FUNCTION_BLOCK FB_Off IMPLEMENTS I_State
VAR_INPUT
	(* Pointer to the ATM Machine*)
	pATM_Machine	: POINTER TO FB_ATM_Machine;
END_VAR
VAR_OUTPUT
END_VAR
VAR
END_VAR

METHOD Cancel : BOOL
END_METHOD

METHOD Card_Ejected : BOOL
END_METHOD

METHOD Card_Inserted : BOOL
END_METHOD

PROPERTY Description : E_StateDescription
GET
Description := E_StateDescription.Off;
END_GET
END_PROPERTY

METHOD Failure : BOOL
END_METHOD

METHOD FB_Init : BOOL
VAR_INPUT
	(* if TRUE, the retain variables are initialized (warm start / cold start)*)
	bInitRetains	: BOOL;
	(* if TRUE, the instance afterwards gets moved into the copy code (online change)*)
	bInCopyCode	: BOOL;
	(* Pointer to the ATM Machine*)
	pATM_Machine	: POINTER TO FB_ATM_Machine;
END_VAR
THIS^.pATM_Machine := pATM_Machine;
END_METHOD

METHOD Op : BOOL
END_METHOD

METHOD Service : BOOL
END_METHOD

METHOD SystemTest_OK : BOOL
END_METHOD

METHOD Turn_Off : BOOL
ADSLOGSTR(ADSLOG_MSGTYPE_LOG, 'Machine is already off!', '');
END_METHOD

METHOD Turn_On : BOOL
ADSLOGSTR(ADSLOG_MSGTYPE_LOG, 'Turning on machine...', '');
pATM_Machine^.SetState(pATM_Machine^.SelfTestState);
END_METHOD

END_FUNCTION_BLOCK

(* stored: Version 1.1.0.1, ProductVersion 3.1.4024.12
   POU FB_Off: Id {77e4ed3a-e16e-0567-22df-368777bf9b32}, SpecialFunc None
   Method Cancel: Id {e3a6cfd6-6764-0ca5-3403-c5b3f56cd495}
   Method Card_Ejected: Id {1c835f53-df5b-0715-2dc8-72b18fbcec93}
   Method Card_Inserted: Id {2426d402-ea1d-097c-3df2-009aefb9d42b}
   Property Description: Id {1255de27-539f-0603-0eb2-fe6707b9ed99}
   Get Get: Id {c0d1b000-d69e-0f80-25cf-a58160038f5f}
   Method Failure: Id {73f3ab78-6cbd-01ce-0db9-9456e1f7b559}
   Method FB_Init: Id {8ffe180d-8c71-0b11-1655-ea2db27e5031}
   Method Op: Id {47dc5cca-e0fc-01e7-28c5-c1653130abde}
   Method Service: Id {6ffc26dc-e3cc-06c8-0c08-82df71cb91b5}
   Method SystemTest_OK: Id {46dc5e76-4dd6-0eac-1ba8-ab13362276aa}
   Method Turn_Off: Id {c404dd17-467e-07fc-3ffd-8d27099a5005}
   Method Turn_On: Id {5f5279f7-f1fa-0345-248c-d404f98f194c} *)
